{attribute 'call_after_init'}
FUNCTION_BLOCK FB_TestSuite_Test EXTENDS TcUnit.FB_TestSuite IMPLEMENTS TcUnit.I_RunnableTestSuite
VAR
    Assert : TcUnit.FB_Assert;

    numberOfTestsZero_TestSuite: UnitTestSuite(0);

    testSuiteRegistersItself_Runner: UnitTestRunner;
    testSuiteRegistersItself_TestSuite: UnitTestSuite(testSuiteRegistersItself_Runner);
    
    runAllTestsWithOneTestSuite_Runner: UnitTestRunner;
    runAllTestsWithOneTestSuite_TestSuite: TestSuiteMock(runAllTestsWithOneTestSuite_Runner);
END_VAR

METHOD FB_init : BOOL
VAR_INPUT
	bInitRetains : BOOL; // if TRUE, the retain variables are initialized (warm start / cold start)
	bInCopyCode : BOOL;  // if TRUE, the instance afterwards gets moved into the copy code (online change)
END_VAR
SUPER^.RegisterTestSuite(THIS^);
END_METHOD

METHOD RunTests : TCUNIT.E_TestSuiteRunState
Test_NumberOfTestsZero();
Test_TestSuiteRegistersItself();
Test_RunAllTestsWithOneTestSuite();

RunTests := TCUNIT.E_TestSuiteRunState.FINISHED;
END_METHOD

METHOD Test_NumberOfTestsZero
VAR
    expected: UINT;
    actual: UINT;
END_VAR
TEST('Test_NumberOfTestsZero');

expected := 0;
actual := numberOfTestsZero_TestSuite.numberOfTests;

Assert.AssertEquals_UINT(expected, actual, 'Number of Tests is non zero');
END_METHOD

METHOD Test_RunAllTestsWithOneTestSuite
VAR
    expected: BOOL;
    actual: BOOL;
END_VAR
TEST('Test_RunAllTestsWithOneTestSuite');

expected := FALSE;
actual := runAllTestsWithOneTestSuite_TestSuite.runAllTestsExecuted;

Assert.AssertEquals_BOOL(expected, actual, 'Test Suite executed even though the runner did not run');

runAllTestsWithOneTestSuite_Runner.runAllTests();

expected := TRUE;
actual := runAllTestsWithOneTestSuite_TestSuite.runAllTestsExecuted;

Assert.AssertEquals_BOOL(expected, actual, 'Test Suite not executed even though the runner ran');
END_METHOD

METHOD Test_TestSuiteRegistersItself
VAR
    expected: UINT;
    actual: UINT;
END_VAR
TEST('Test_TestSuiteRegistersItself');

expected := 1;
actual := testSuiteRegistersItself_Runner.numberOfTestSuites;

Assert.AssertEquals_UINT(expected, actual, 'Test Suite did not register itself');
END_METHOD

END_FUNCTION_BLOCK

(* stored: Version 1.1.0.1, ProductVersion 3.1.4022.12
   POU FB_TestSuite_Test: Id {d2c06896-6e3c-40b1-9e7c-b4cc8df87908}, SpecialFunc None
   Method FB_init: Id {1badc6ad-ade3-4405-9c9a-df88f28d0da4}
   Method RunTests: Id {dd012402-76f5-4bcc-bd36-986590cd1111}
   Method Test_NumberOfTestsZero: Id {cd3b711a-9f58-40f4-8711-9a9ecbf8282a}
   Method Test_RunAllTestsWithOneTestSuite: Id {1b323fd8-3565-44ad-8ceb-2b26a6fa02c2}
   Method Test_TestSuiteRegistersItself: Id {b71098b5-ba04-4e73-a831-e0685a1e4a93} *)
